FUNCTION_BLOCK FB_FileHandler
VAR_INPUT
	sNetId: T_AmsNetId;
	sPathName: T_MaxString;
	
END_VAR
VAR_OUTPUT
END_VAR
VAR
	fbFileOpen : FB_FileOpen;
	fbFileClose : FB_FileClose;
	fbFileSeek : FB_FileSeek;
	fbFileTell : FB_FileTell;
	
	
	stepGetFileSize : INT;
	_hFile: UINT;
	
	
END_VAR

fbFileOpen(
	sNetId:= sNetId, 
	sPathName:= sPathName, 
	nMode:= FOPEN_MODEREAD OR FOPEN_MODEPLUS OR FOPEN_MODEBINARY, 
	ePath:= PATH_GENERIC, 
	bExecute:= , 
	tTimeout:= DEFAULT_ADS_TIMEOUT, 
	bBusy=> , 
	bError=> , 
	nErrId=> , 
	hFile=> _hFile);

METHOD GetFileSize : UDINT
VAR_INPUT
END_VAR
CASE stepGetFileSize OF
0:
	





END_CASE
END_METHOD

METHOD Open : BOOL
VAR_INPUT
END_VAR

fbFileOpen(bExecute := TRUE);
IF  NOT fbFileOpen.bBusy AND NOT fbFileOpen.bError THEN
	Open := TRUE;
END_IF
END_METHOD

END_FUNCTION_BLOCK

(* stored: Version 1.1.0.1, ProductVersion 3.1.4024.12
   POU FB_FileHandler: Id {2c918a86-39ee-4304-b138-735a315529dc}, SpecialFunc None
   Method GetFileSize: Id {9b179687-9024-4361-8d36-60346d911616}
   Method Open: Id {2dc6a26f-5d67-458f-9aea-067323bf8136} *)
